FUNCTION_BLOCK RefactoringLongReal
VAR_INPUT
	I_Percentage:				LREAL;
	I_MaximumValue:					LREAL;
END_VAR
VAR_OUTPUT
	Q_Result:					LREAL;
END_VAR
VAR
END_VAR

Q_Result:=(I_Percentage*I_MaximumValue)/100;

END_FUNCTION_BLOCK

(* stored: Version 1.1.0.1, ProductVersion 3.1.4022.18
   POU RefactoringLongReal: Id {ae7cb5c4-f664-44e3-b234-78d022668a38}, SpecialFunc None *)
